(* IEC 61131-3 sources: axftcmlib/src/Motor, 4 files *)

(* ---- IMotor.st ---- *)
NAMESPACE Simatic.Ax.axftcmlib.Motion
    // This interface provides methods to control a bidirectional  motor.
    INTERFACE IMotorBiDiretional
        ///Starts the Motor with a given direction and velocity
        METHOD Move
            VAR_INPUT
                velocity : LREAL;
                direction : Direction;
            END_VAR
        END_METHOD
        ///Stops every movement of the Motor
        METHOD Halt
        END_METHOD
    END_INTERFACE
END_NAMESPACE

(* ---- Motor.st ---- *)
USING Simatic.Ax.IO.Output;
USING Simatic.Ax.axftcmlib;

NAMESPACE Simatic.Ax.axftcmlib.Motion

    ///Class for creating a basic Motor
    /// It supports two directions
    /// It is used to power the axis
    CLASS MotorFT IMPLEMENTS IMotor
        VAR PUBLIC
            Forward : IBinOutput;
            Reverse : IBinOutput;
        END_VAR
        VAR PROTECTED
        END_VAR
        ///Starts the Motor with a given direction and velocity
        METHOD PUBLIC Move
            VAR_INPUT
                velocity : LREAL;
                direction : Direction;
            END_VAR
            IF (direction = Direction#PositiveDirection) THEN
                Forward.SetOn();
                Reverse.SetOff();
            ELSE
                Reverse.SetOn();
                Forward.SetOff();
            END_IF;
            ;
        END_METHOD
        ///Stops every movement of the Motor
        METHOD PUBLIC Halt
            Reverse.SetOff();
            Forward.SetOff();
            ;
        END_METHOD
    END_CLASS

END_NAMESPACE

(* ---- MotorBiDirectional.st ---- *)
USING Simatic.Ax.IO.Output;
USING Simatic.Ax.axftcmlib;

NAMESPACE Simatic.Ax.axftcmlib.Motion

    ///Class for creating a basic Motor
    /// It supports two directions
    /// It is used to power the axis
    CLASS MotorFT
        IMPLEMENTS IMotorBiDiretional
        VAR PUBLIC
            Forward : IBinOutput;
            Reverse : IBinOutput;
        END_VAR
        VAR PROTECTED
        END_VAR
        ///Starts the Motor with a given direction and velocity

        METHOD PUBLIC Move
            VAR_INPUT
                velocity : LREAL;
                direction : Direction;
            END_VAR
            IF (direction = Direction#PositiveDirection) THEN
                IF (Forward <> NULL) THEN
                    Forward.SetOn();
                END_IF;
                IF (Reverse <> NULL) THEN
                    Reverse.SetOff();
                END_IF;
            ELSE
                IF (Forward <> NULL) THEN
                    Forward.SetOff();
                END_IF;
                IF (Reverse <> NULL) THEN
                    Reverse.SetOn();
                END_IF;
            END_IF;
            ;
        END_METHOD
        ///Stops every movement of the Motor

        METHOD PUBLIC Halt
              IF (Forward <> NULL) THEN
                    Forward.SetOff();
                END_IF;
                IF (Reverse <> NULL) THEN
                    Reverse.SetOff();
                END_IF;
            ;
        END_METHOD
    END_CLASS

END_NAMESPACE

(* ---- MotorUniDirectional.st ---- *)
USING Simatic.Ax.IO.Output;
USING Simatic.Ax.axftcmlib;

NAMESPACE Simatic.Ax.axftcmlib.Motion

    ///Class for creating a basic Motor
    /// It supports two directions
    /// It is used to power the axis
    CLASS MotorUniDirectional IMPLEMENTS IMotor
        VAR PUBLIC
            Forward : IBinOutput;
        END_VAR
        VAR PROTECTED
        END_VAR
        ///Starts the Motor with a given direction and velocity
        METHOD PUBLIC Move
            VAR_INPUT
                velocity : LREAL;
            END_VAR
            Forward.SetOn();
            ;
        END_METHOD
        ///Stops every movement of the Motor
        METHOD PUBLIC Halt
            Forward.SetOff();
            ;
        END_METHOD
    END_CLASS

END_NAMESPACE
